INTERFACE EventManager

METHOD ClearAll
VAR_INPUT
END_VAR
END_METHOD

END_INTERFACE

(* stored: Version 1.1.0.1
   Itf EventManager: Id {e6aa0918-6d48-0701-2ddd-9942b00b9e2a}
   Method ClearAll: Id {86cd8969-20c0-05a5-2c6f-a7c3cf2340eb} *)
